{attribute 'qualified_only'}
VAR_GLOBAL
	
END_VAR

(* stored: Version 1.1.0.1, ProductVersion 3.1.4024.16
   GVL TRIAL: Id {08abc386-7020-4c44-ab9f-f92c3b99c3e8} *)
